// SIMATIC STEP 7 (V5.x) project TEMA 8 EJERCICIIO 2
// CPU: CPU313 C-2 DP(1)
// station: P_ADR_BUS
// station: Hardware
// station: Equipo SIMATIC 300
// program: Programa S7(1)

SYMBOL_TABLE
""		
""		
""		
""		
"FLANCO"	DB 1	DB 1
"MANIOBRA"	DB 2	DB 2
"P PARO"	I 0.0	BOOL
"P DERECHAS"	I 0.1	BOOL
"P IZQUIERDAS"	I 0.2	BOOL
"R TERMICO"	I 0.3	BOOL
"LED PARO"	Q 0.0	BOOL
"LINEA DERECHAS"	Q 0.1	BOOL
"LINEA IZQUIERDAS"	Q 0.2	BOOL
"ESTRELLA"	Q 0.3	BOOL
"TRIANGULO"	Q 0.4	BOOL
"LED DERECHAS"	Q 0.5	BOOL
"LED IZQUIERDAS"	Q 0.6	BOOL
"LED AVERIA"	Q 0.7	BOOL
"VAT_1"	VAT 1	
END_SYMBOL_TABLE

DATA_BLOCK "FLANCO"	// DB 1
VERSION : 0.1
  STRUCT
   MARCA0 : BOOL ;
   MARCA1 : BOOL ;
   MARCA2 : BOOL ;
   MARCA3 : BOOL ;
   MARCA4 : BOOL ;
   MARCA5 : BOOL ;
   MARCA6 : BOOL ;
   MARCA7 : BOOL ;
   MARCA10 : BOOL ;
   MARCA11 : BOOL ;
   MARCA12 : BOOL ;
   MARCA13 : BOOL ;
   MARCA14 : BOOL ;
   MARCA15 : BOOL ;
   MARCA16 : BOOL ;
   MARCA17 : BOOL ;
   MARCA20 : BOOL ;
   MARCA21 : BOOL ;
   MARCA22 : BOOL ;
   MARCA23 : BOOL ;
   MARCA24 : BOOL ;
   MARCA25 : BOOL ;
   MARCA26 : BOOL ;
   MARCA27 : BOOL ;
  END_STRUCT ;	
BEGIN
END_DATA_BLOCK

DATA_BLOCK "MANIOBRA"	// DB 2
VERSION : 0.1
  STRUCT
   MARCA0 : BOOL ;
   MARCA1 : BOOL ;
   MARCA2 : BOOL ;
   MARCA3 : BOOL ;
   MARCA4 : BOOL ;
   MARCA5 : BOOL ;
   MARCA6 : BOOL ;
   MARCA7 : BOOL ;
  END_STRUCT ;	
BEGIN
END_DATA_BLOCK

ORGANIZATION_BLOCK OB 1
TITLE = "Main Program Sweep (Cycle)"
//ARRANQUE ESTRELLA -TRIANGULO CON INVERSION DE GIRO
VERSION : 0.1
VAR_TEMP
  OB1_EV_CLASS : BYTE ;	//Bits 0-3 = 1 (Coming event), Bits 4-7 = 1 (Event class 1)
  OB1_SCAN_1 : BYTE ;	//1 (Cold restart scan 1 of OB 1), 3 (Scan 2-n of OB 1)
  OB1_PRIORITY : BYTE ;	//Priority of OB Execution
  OB1_OB_NUMBR : BYTE ;	//1 (Organization block 1, OB1)
  OB1_RESERVED_1 : BYTE ;	//Reserved for system
  OB1_RESERVED_2 : BYTE ;	//Reserved for system
  OB1_PREV_CYCLE : INT ;	//Cycle time of previous OB1 scan (milliseconds)
  OB1_MIN_CYCLE : INT ;	//Minimum cycle time of OB1 (milliseconds)
  OB1_MAX_CYCLE : INT ;	//Maximum cycle time of OB1 (milliseconds)
  OB1_DATE_TIME : DATE_AND_TIME ;	//Date and time OB1 started
END_VAR
BEGIN
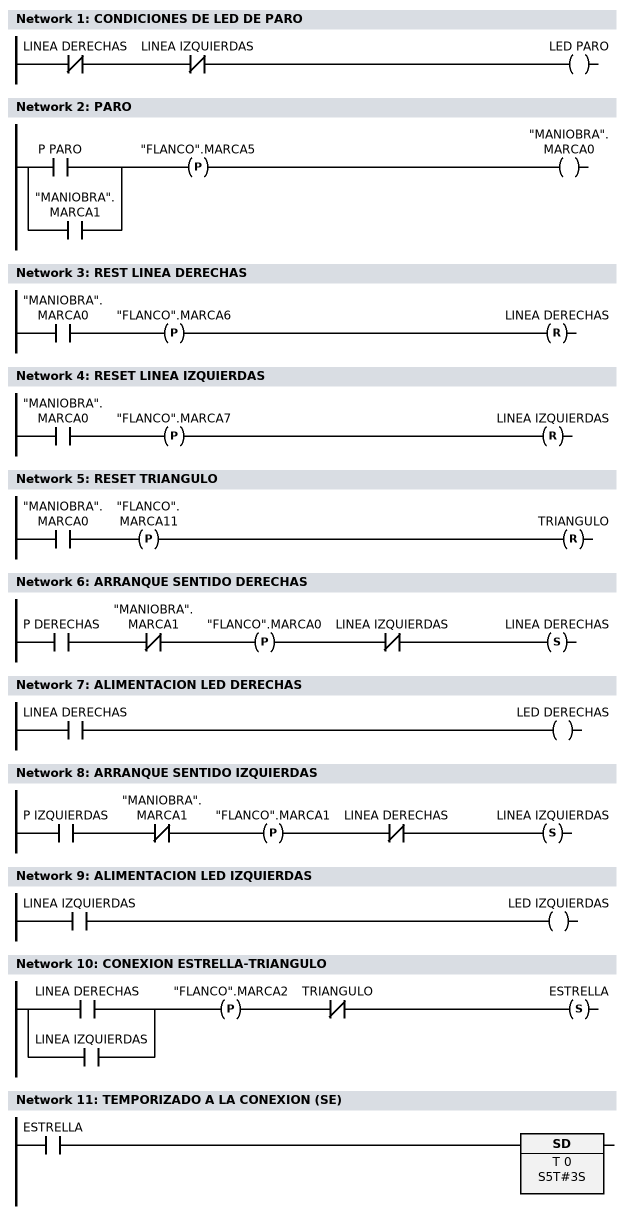
NETWORK
TITLE = CONDICIONES DE LED DE PARO
//ESTADO INICIAL REPOSO LED ENCENDIDA 
      AN    "LINEA DERECHAS";
      AN    "LINEA IZQUIERDAS";
      =     "LED PARO";
NETWORK
TITLE = PARO
//RESETEA BOBINAS TANTO DE DERECHAS COMO IZQUIERDAS
      A(;
      O     "P PARO";
      O     "MANIOBRA".MARCA1;
      );
      FP    "FLANCO".MARCA5;
      =     "MANIOBRA".MARCA0;
NETWORK
TITLE = REST LINEA DERECHAS
      A     "MANIOBRA".MARCA0;
      FP    "FLANCO".MARCA6;
      R     "LINEA DERECHAS";
NETWORK
TITLE = RESET LINEA IZQUIERDAS
      A     "MANIOBRA".MARCA0;
      FP    "FLANCO".MARCA7;
      R     "LINEA IZQUIERDAS";
NETWORK
TITLE = RESET TRIANGULO
      A     "MANIOBRA".MARCA0;
      FP    "FLANCO".MARCA11;
      R     "TRIANGULO";
NETWORK
TITLE = ARRANQUE SENTIDO DERECHAS 
//PULASADOR DERECHAS ALIMENTA LINEA DERECHAS
      A     "P DERECHAS";
      AN    "MANIOBRA".MARCA1;
      FP    "FLANCO".MARCA0;
      AN    "LINEA IZQUIERDAS";
      S     "LINEA DERECHAS";
NETWORK
TITLE = ALIMENTACION LED DERECHAS
      A     "LINEA DERECHAS";
      =     "LED DERECHAS";
NETWORK
TITLE = ARRANQUE SENTIDO IZQUIERDAS
//PULSADOR IZQUIERDAS ALIMENTA LINEA IZQUIERDAS
      A     "P IZQUIERDAS";
      AN    "MANIOBRA".MARCA1;
      FP    "FLANCO".MARCA1;
      AN    "LINEA DERECHAS";
      S     "LINEA IZQUIERDAS";
NETWORK
TITLE = ALIMENTACION LED IZQUIERDAS
      A     "LINEA IZQUIERDAS";
      =     "LED IZQUIERDAS";
NETWORK
TITLE = CONEXION ESTRELLA-TRIANGULO
//ACTIVACION CONEXION ESTRELLA ;CONTACTO AUXILIAR DE A0.1 Y A0.2
//
      A(;
      O     "LINEA DERECHAS";
      O     "LINEA IZQUIERDAS";
      );
      FP    "FLANCO".MARCA2;
      AN    "TRIANGULO";
      S     "ESTRELLA";
NETWORK
TITLE = TEMPORIZADO A LA CONEXION (SE)
//ACTIVACION TEMPORIZADOR 3 SEG.
      A     "ESTRELLA";
      L     S5T#3S;
      SD    T 0;
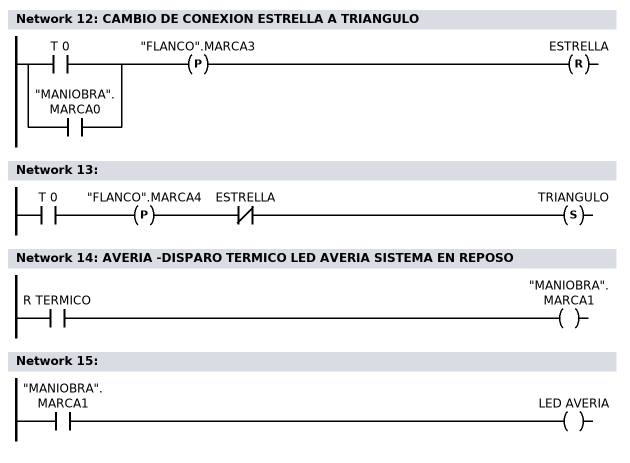
NETWORK
TITLE = CAMBIO DE CONEXION ESTRELLA A TRIANGULO
//CONTACTO TEMPORIZADO DESCONECTA ESTRELLA 
      A(;
      O     T 0;
      O     "MANIOBRA".MARCA0;
      );
      FP    "FLANCO".MARCA3;
      R     "ESTRELLA";
NETWORK
TITLE =
//CONECTA TRIANGULO
      A     T 0;
      FP    "FLANCO".MARCA4;
      AN    "ESTRELLA";
      S     "TRIANGULO";
NETWORK
TITLE = AVERIA -DISPARO TERMICO LED AVERIA SISTEMA EN REPOSO
//CONTACTACTO AUXILIAR DE MANIOBRA 1
      A     "R TERMICO";
      =     "MANIOBRA".MARCA1;
NETWORK
TITLE =
//ENCENDIO LED AVERIA 
      A     "MANIOBRA".MARCA1;
      =     "LED AVERIA";
END_ORGANIZATION_BLOCK

ORGANIZATION_BLOCK OB 80
TITLE = "Cycle Time Fault"
VERSION : 0.1
VAR_TEMP
  OB80_EV_CLASS : BYTE ;	//16#35, Event class 3, Entering event state, Internal fault event
  OB80_FLT_ID : BYTE ;	//16#XX, Fault identifcation code
  OB80_PRIORITY : BYTE ;	//Priority of OB Execution
  OB80_OB_NUMBR : BYTE ;	//80 (Organization block 80, OB80)
  OB80_RESERVED_1 : BYTE ;	//Reserved for system
  OB80_RESERVED_2 : BYTE ;	//Reserved for system
  OB80_ERROR_INFO : WORD ;	//Error information on event
  OB80_ERR_EV_CLASS : BYTE ;	//Class of event causing error
  OB80_ERR_EV_NUM : BYTE ;	//Number of event causing error
  OB80_OB_PRIORITY : BYTE ;	//Priority of OB causing error
  OB80_OB_NUM : BYTE ;	//Number of OB causing error
  OB80_DATE_TIME : DATE_AND_TIME ;	//Date and time OB80 started
END_VAR
BEGIN
// (block stored without names or comments; labels and parameter names are numbered)
END_ORGANIZATION_BLOCK

ORGANIZATION_BLOCK OB 81
TITLE = "Power Supply Fault"
VERSION : 0.1
VAR_TEMP
  OB81_EV_CLASS : BYTE ;	//16#39, Event class 3, Entering event state, Internal fault event
  OB81_FLT_ID : BYTE ;	//16#XX, Fault identifcation code
  OB81_PRIORITY : BYTE ;	//Priority of OB Execution
  OB81_OB_NUMBR : BYTE ;	//81 (Organization block 81, OB81)
  OB81_RESERVED_1 : BYTE ;	//Reserved for system
  OB81_RESERVED_2 : BYTE ;	//Reserved for system
  OB81_RACK_CPU : WORD ;	//see online help (F1)
  OB81_RESERVED_3 : BYTE ;	//Reserved for system
  OB81_RESERVED_4 : BYTE ;	//Reserved for system
  OB81_RESERVED_5 : BYTE ;	//Reserved for system
  OB81_RESERVED_6 : BYTE ;	//Reserved for system
  OB81_DATE_TIME : DATE_AND_TIME ;	//Date and time OB81 started
END_VAR
BEGIN
// (block stored without names or comments; labels and parameter names are numbered)
END_ORGANIZATION_BLOCK
